// TIA Portal V17 export
// export: Created 2024-09-02T12:50:26.8335936Z, ExportSetting WithDefaults, DisplayName Totally Integrated Automation Portal, DisplayVersion V17, DisplayName TIA Portal Openness, DisplayVersion V17, DisplayName TIA Portal Version Control Interface, DisplayVersion V17, DisplayName STEP 7 Professional, DisplayVersion V17, DisplayName STEP 7 Safety, DisplayVersion V17, DisplayName WinCC Professional, DisplayVersion V17
TYPE "af_MGB"
// stored: IsFailsafeCompliant true
   STRUCT
      TürÖffnen : Bool;   // Profisafe - Magnet Tür öffnen / Profisafe - magnet open door
      "res5.1" : Bool;   // Profisafe - Reserve
      "res5.2" : Bool;   // Profisafe - Reserve
      "res5.3" : Bool;   // Profisafe - Reserve
      "res5.4" : Bool;   // Profisafe - Reserve
      "res5.5" : Bool;   // Profisafe - Reserve
      "res5.6" : Bool;   // Profisafe - Reserve
      "res5.7" : Bool;   // Profisafe - Reserve
      "res6.0" : Bool;   // Profisafe - Reserve
      "res6.1" : Bool;   // Profisafe - Reserve
      "res6.2" : Bool;   // Profisafe - Reserve
      "res6.3" : Bool;   // Profisafe - Reserve
      "res6.4" : Bool;   // Profisafe - Reserve
      "res6.5" : Bool;   // Profisafe - Reserve
      "res6.6" : Bool;   // Profisafe - Reserve
      "res6.7" : Bool;   // Profisafe - Reserve
      "res7.0" : Bool;   // Profisafe - Reserve
      "res7.1" : Bool;   // Profisafe - Reserve
      "res7.2" : Bool;   // Profisafe - Reserve
      "res7.3" : Bool;   // Profisafe - Reserve
      "res7.4" : Bool;   // Profisafe - Reserve
      "res7.5" : Bool;   // Profisafe - Reserve
      "res7.6" : Bool;   // Profisafe - Reserve
      "res7.7" : Bool;   // Profisafe - Reserve
      "res8.0" : Bool;   // Profisafe - Reserve
      "res8.1" : Bool;   // Profisafe - Reserve
      "res8.2" : Bool;   // Profisafe - Reserve
      "res8.3" : Bool;   // Profisafe - Reserve
      "res8.4" : Bool;   // Profisafe - Reserve
      "res8.5" : Bool;   // Profisafe - Reserve
      "res8.6" : Bool;   // Profisafe - Reserve
      "res8.7" : Bool;   // Profisafe - Reserve
      "res9.0" : Bool;   // Profisafe - Reserve
      "res9.1" : Bool;   // Profisafe - Reserve
      "res9.2" : Bool;   // Profisafe - Reserve
      "res9.3" : Bool;   // Profisafe - Reserve
      "res9.4" : Bool;   // Profisafe - Reserve
      "res9.5" : Bool;   // Profisafe - Reserve
      "res9.6" : Bool;   // Profisafe - Reserve
      "res9.7" : Bool;   // Profisafe - Reserve
      "res10.0" : Bool;   // Profisafe - Reserve
      "res10.1" : Bool;   // Profisafe - Reserve
      "res10.2" : Bool;   // Profisafe - Reserve
      "res10.3" : Bool;   // Profisafe - Reserve
      "res10.4" : Bool;   // Profisafe - Reserve
      "res10.5" : Bool;   // Profisafe - Reserve
      "res10.6" : Bool;   // Profisafe - Reserve
      "res10.7" : Bool;   // Profisafe - Reserve
   END_STRUCT;
END_TYPE
